{attribute 'strict'}
TYPE E_XPU_CTRL :
(
  XTS_CMD_NULL,
  XTS_CMD_INIT                  := 10,
  //XTS_CMD_READ_STN_CONFIG       := 20,
  XTS_IDLE                      := 30
)UINT;
END_TYPE

(* stored: Version 1.1.0.1
   DUT E_XPU_CTRL: Id {f74e9a0c-327d-4efd-89c3-6459427caa15} *)
